// TwinCAT 3 PLC project PLC_LocateEdge
// ProgramVersion: 3.1.4023.0
// libraries:
//   Tc2_Standard, * (Beckhoff Automation GmbH)
//   Tc2_System, * (Beckhoff Automation GmbH)
//   Tc2_Utilities, * (Beckhoff Automation GmbH)
//   Tc3_Module, * (Beckhoff Automation GmbH)
//   Tc3_Vision, * (Beckhoff Automation GmbH)
// project tree:
//   DUTs/ ST_DimBase.TcDUT
//   GVLs/ GVL.TcGVL
//   / PlcTask.TcTTO, Vision_Job_Task_0.TcTTO
//   POUs/ FB_Camera.TcPOU, FB_MinAvgMax.TcPOU, F_Angle.TcPOU, F_Distance.TcPOU, F_DimDraw.TcPOU, MAIN.TcPOU, MAIN_VISION.TcPOU
// real-time tasks:
//   TASK PlcTask: cycle T#2ms, priority 4, ADS port 351
//   TASK VnTask ImgAcq (FileSource1): cycle T#5ms, priority 8, ADS port 350
//   TASK Vision Job Task 1: cycle default, priority 1
//   TASK Vision Job Task 0: cycle T#200000us, priority 10, ADS port 352

CONFIGURATION PLC_LocateEdge
    RESOURCE PLC ON TwinCAT3
        TASK PlcTask(INTERVAL := T#2ms, PRIORITY := 4);
        TASK Vision_Job_Task_0(INTERVAL := T#200000us, PRIORITY := 10);
        PROGRAM MAIN WITH PlcTask : MAIN;
        PROGRAM MAIN_VISION WITH Vision_Job_Task_0 : MAIN_VISION;
    END_RESOURCE
END_CONFIGURATION

// ---- DUTs/ST_DimBase.TcDUT
TYPE ST_DimBase :
STRUCT
	// Config
	name : STRING(255);
	
	// Must be set. Default values will return errors
	pFrom : TcVnPoint2_REAL := [-1, -1];
	pTo1 : TcVnPoint2_REAL := [-1, -1];
	pTo2 : TcVnPoint2_REAL := [-1, -1]; // Used for angle
	lines : UDINT := 0;
	
	// Can use defaults
	dir : ETcVnEdgeDirection := TCVN_ED_LIGHT_TO_DARK;
	minStr : REAL := 50;
	lineDist : REAL := 1;
	maxThick : UDINT := 10;
	gap : REAL := 0;
	precision : REAL := 0.0001; // 0.01 - 0.0001 only used for ERF/Gaussian
	subpix : UDINT := 1000; // 5-20 for INTER, 50-100 for ERF/Gaussian
	invDir : BOOL := FALSE;
	algorithm : ETcVnEdgeDetectionAlgorithm := TCVN_EDA_APPROX_ERF;
	degrees : BOOL := TRUE; // Used for angle
	
	// Results
	result : REAL;
	et : DINT; // Elapsed time in us
	complete : UDINT;
	results : ITcVnContainer; // Used for distance
	edgeFrom : ITcVnContainer;
	edgeTo : ITcVnContainer;
	lineFrom : TcVnVector4_LREAL;
	lineTo : TcVnVector4_LREAL;
END_STRUCT
END_TYPE

// ---- GVLs/GVL.TcGVL
VAR_GLOBAL
	camera : FB_Camera;
	dimDist : ARRAY [0..4] OF ST_DimBase := [
		(name:='d201', pFrom:=[115, 1290], pTo1:=[640, 1290], gap:=-1, lines:=291, lineDist:=3),
		(name:='d209', pFrom:=[245, 795], pTo1:=[245, 1770], gap:=-1, lines:=49, lineDist:=4),
		(name:='d222', pFrom:=[760, 875], pTo1:=[760, 1700], gap:=-1, lines:=45, lineDist:=4),
		(name:='od', pFrom:=[2260, 970], pTo1:=[2260, 1650], gap:=-1, lines:=121, lineDist:=4),
		(name:='gripper', pFrom:=[860, 450], pTo1:=[1850, 450], gap:=-1, lines:=161, lineDist:=5)
	];
END_VAR

// ---- POUs/MAIN.TcPOU
PROGRAM MAIN
VAR
	res : ARRAY [0..4] OF FB_MinAvgMax;
	ets : ARRAY [0..5] OF FB_MinAvgMax;
	total_et : DINT;
	test: BOOL;
	ii: INT;
	state: INT;
	cnt : INT;
	test2: BOOL;
	
	avg : LREAL;
	avg1 : TcVnVector2_LREAL;
	avg2 : TcVnVector2_LREAL;
	size1 : ULINT;
	size2 : ULINT;
	size3 : ULINT;
	
	idx : INT;
	arr1 : ARRAY [0..500] OF TcVnVector2_REAL;
	arr2 : ARRAY [0..500] OF TcVnVector2_REAL;
	arr3 : ARRAY [0..500] OF REAL;
END_VAR


IF test THEN
	test := FALSE;
	camera.trig();
END_IF

IF test2 THEN
	test2 := FALSE;
	F_VN_ContainerAverage(dimDist[idx].results, avg, S_OK);
	F_VN_ContainerAverageElementwise2(dimDist[idx].edgeFrom, avg1, S_OK);
	F_VN_ContainerAverageElementwise2(dimDist[idx].edgeTo, avg2, S_OK);
	
	F_VN_ExportContainerSize(dimDist[idx].edgeFrom, size1, S_OK);
	F_VN_ExportContainerSize(dimDist[idx].edgeTo, size2, S_OK);
	F_VN_ExportContainerSize(dimDist[idx].results, size3, S_OK);
	
	F_VN_ExportContainer(dimDist[idx].edgeFrom, ADR(arr1), SIZEOF(arr1), s_ok);
	F_VN_ExportContainer(dimDist[idx].edgeTo, ADR(arr2), SIZEOF(arr2), s_ok);
	F_VN_ExportContainer(dimDist[idx].results, ADR(arr3), SIZEOF(arr3), s_ok);
END_IF

CASE state OF
	10:
		camera.trig();
		state := 11;
	11:
		IF NOT camera.busy THEN
			total_et := 0;
			FOR ii := 0 TO 4 DO
				res[ii](IN:=dimDist[ii].result);
				ets[ii](IN:=dimDist[ii].et);
				total_et := total_et + dimDist[ii].et;
			END_FOR
			ets[5](IN:=total_et);
			cnt := cnt + 1;
			IF cnt < 100 THEN
				state := 10;
			ELSE
				cnt := 0;
				state := 0;
			END_IF
		END_IF
	12:
		FOR ii := 0 TO 4 DO
			res[ii].reset();
			ets[ii].reset();
		END_FOR
		ets[5].reset();
		state := 0;
END_CASE

END_PROGRAM

// ---- POUs/FB_MinAvgMax.TcPOU
FUNCTION_BLOCK FB_MinAvgMax
VAR_INPUT
	IN		: LREAL;
END_VAR
VAR_OUTPUT
	mini	: LREAL := 1.7976931348623158E308;
	avge	: LREAL;
	maxi	: LREAL := -1.7976931348623158E308;
END_VAR
VAR
	nums	: LREAL;
END_VAR

IF IN > maxi THEN
	maxi := IN;
END_IF
IF IN < mini THEN
	mini := IN;
END_IF

nums := nums + 1;
avge := avge + (IN - avge) / nums;

METHOD reset : BOOL
VAR_INPUT
END_VAR

mini := +1.7976931348623158E308;
maxi := -1.7976931348623158E308;
avge := 0;
nums := 0;
END_METHOD

END_FUNCTION_BLOCK

// ---- POUs/MAIN_VISION.TcPOU
PROGRAM MAIN_VISION
VAR
END_VAR


camera(dims := dimDist);

END_PROGRAM

// ---- POUs/FB_Camera.TcPOU
FUNCTION_BLOCK FB_Camera
VAR_IN_OUT
	dims : ARRAY [*] OF ST_DimBase;
END_VAR
VAR_OUTPUT
	busy : BOOL;
	ET : DINT;
END_VAR
VAR
	hr : HRESULT;
	hrFunc : HRESULT;
	hrWD : HRESULT;
	
	camera : FB_VN_SimpleCameraControl;
	camState : ETcVnCameraState;
	
	imgIn : ITcVnImage;
	imgInDisp : ITcVnDisplayableImage;
	imgOut : ITcVnImage;
	imgOutDisp : ITcVnDisplayableImage;
	
	state : INT;
	preempt : DINT;
	remain : DINT;
	complete : UDINT;
	ii : DINT;
	upper : DINT;
	lower : DINT;
	trigger : BOOL;
	cycleCnt : INT;
	old: INT;
	hr1:HRESULT;
	hr2:HRESULT;
END_VAR


camState := camera.GetState();
CASE state OF
	0:
		lower := LOWER_BOUND(dims, 1);
		upper := UPPER_BOUND(dims, 1);
		// Allow 1 ms for other items in task before and after vision
		preempt := TO_DINT(_TaskInfo[GETCURTASKINDEXEX()].CycleTime / 10) - 1000;
		IF preempt < 1000 THEN
			// Task cycle time is 1ms or less. Will not work.
			state := -1;
		ELSE
			state := 1000;
		END_IF
	1000:
		busy := FALSE;
		CASE camState OF
			TCVN_CS_INITIAL, TCVN_CS_OPENING, TCVN_CS_OPENED, TCVN_CS_STARTACQUISITION:
				hr := camera.StartAcquisition();
			TCVN_CS_Error:
				state := -1;
		END_CASE
	1010:
		CASE camState OF
			TCVN_CS_TRIGGERING:
				// If getting 16#98110712 the source likely has trigger disabled
				hr1 := camera.TriggerImage();
			TCVN_CS_ACQUIRING:
				IF trigger THEN
					hr2 := camera.TriggerImage();
					IF succeeded(hr2) THEN
						trigger := FALSE;
					END_IF
				ELSE
					hr := camera.GetCurrentImage(imgIn);
					IF SUCCEEDED(hr) AND_THEN imgIn <> 0 THEN
						ii := lower;
						ET := 0;
						cycleCnt := 0;
						state := 1020;
					END_IF
				END_IF
			TCVN_CS_ERROR:
				state := -1;
		END_CASE
	1020:
		remain := preempt; // Reset remain on each new cycle
		cycleCnt := cycleCnt + 1;
		FOR ii := ii TO upper DO
			hrWD := F_VN_StartRelWatchdog(remain, S_OK);
			// If returns 16#71A Task Watchdog Stack not enabled
			IF dims[ii].pTo2[0] = -1 THEN
				// pTo2 not used in Distance measurement
				hrFunc := F_Distance(dims[ii], imgIn);
			ELSE
				// But it is used in angle measurement
				hrFunc := F_Angle(dims[ii], imgIn);
			END_IF
			hrWD := F_VN_StopWatchdog(hrWD, nFractionProcessed=>complete, tRest=>remain);
			IF FAILED(hrFunc) OR_ELSE FAILED(hrWD) THEN
				// Send failed message
				// Will move on to other inspections and this one is ignored
			END_IF
			dims[ii].et := (cycleCnt * preempt) - ET - remain;
			dims[ii].complete := complete;
			ET := ET + dims[ii].et;
			IF complete <> 100 AND_THEN SUCCEEDED(hrFunc) THEN
				// Try calculation again in new cycle if not complete, but also not errored
				// Watchdog likely stopped it before completion
				EXIT;
			ELSIF ii = upper THEN
				// All calculations completed
				state := 1030;
				EXIT;
			ELSIF dims[ii+1].et > remain OR_ELSE (dims[ii+1].et = 0 AND_THEN remain < 1000) THEN
				// If the calculation was already done check its elapsed time larger than remain
				// If first time doing then try if more then 1ms remain otherwise start on new cycle
				ii := ii + 1;
				EXIT;
			END_IF
		END_FOR
	1030:
		hr := F_VN_ConvertColorSpace(imgIn, imgOut, TCVN_CST_GRAY_TO_RGB, hr);
		FOR ii := lower TO upper DO
			F_DimDraw(dims[ii], imgOut);
		END_FOR
		
		hr := F_VN_TransformIntoDisplayableImage(imgIn, imgInDisp, S_OK);
		hr := F_VN_TransformIntoDisplayableImage(imgOut, imgOutDisp, S_OK);
		state := 1000;
	-1000:
		// If stays in error then not linked to file/device
		// Check instance symbol initialization
		camera.Reset();
		IF camState <> TCVN_CS_ERROR THEN
			state := 0;
		END_IF
END_CASE

METHOD trig : BOOL
VAR_INPUT
END_VAR

IF state = 1000 AND_THEN camState = TCVN_CS_ACQUIRING AND_THEN NOT busy THEN
	busy := TRUE;
	ET := 0;
	trigger := TRUE;
	state := 1010;
END_IF
END_METHOD

END_FUNCTION_BLOCK

// ---- POUs/F_Distance.TcPOU
FUNCTION F_Distance : HRESULT
VAR_INPUT
	dim : REFERENCE TO ST_DimBase;
	img : ITcVnImage;
END_VAR


IF dim.gap < 0 THEN
	// If gap less than zero auto calculate based on largest diff between x/y and set to 80%
	// Helps reduce computation time
	dim.gap := MAX(ABS(dim.pTo1[0] - dim.pFrom[0]), ABS(dim.pTo1[1] - dim.pFrom[1])) * 0.8;
END_IF

F_Distance := F_VN_MeasureEdgeDistanceExp(
	ipSrcImage:=img,
	fAvgDistance:=dim.result,
	aStartPoint:=dim.pFrom,
	aEndPoint:=dim.pTo1,
	eEdgeDirection:=dim.dir,
	fMinStrength:=dim.minStr,
	nSearchLines:=dim.lines,
	fSearchLineDist:=dim.lineDist,
	nMaxThickness:=dim.maxThick,
	bInvertSearchDirection:=dim.invDir,
	fSearchGap:=dim.gap,
	nSubpixelsIterations:=dim.subpix,
	fApproxPrecision:=dim.precision,
	eAlgorithm:=dim.algorithm,
	ipEdgePoints1:=dim.edgeFrom,
	ipEdgePoints2:=dim.edgeTo,
	ipDistances:=dim.results,
	hrPrev:=S_OK
);

END_FUNCTION

// ---- POUs/F_Angle.TcPOU
FUNCTION F_Angle : HRESULT
VAR_INPUT
	dim : REFERENCE TO ST_DimBase;
	img : ITcVnImage;
END_VAR


F_Angle := F_VN_MeasureAngleBetweenEdgesExp(
	ipSrcImage:= img,
	fAngle:= dim.result,
	aInnerPoint:= dim.pFrom,
	aOuterPoint1:= dim.pTo1,
	aOuterPoint2:= dim.pTo2,
	eEdgeDirection:= dim.dir,
	fMinStrength:= dim.minStr,
	nSearchLines:= dim.lines,
	fSearchLineDist:= dim.lineDist,
	nMaxThickness:= dim.maxThick,
	bInvertSearchDirection:= dim.invDir,
	nSubpixelsIterations:= dim.subpix,
	bAngleInDegrees:= dim.degrees,
	fApproxPrecision:= dim.precision,
	eAlgorithm:= dim.algorithm,
	ipEdgePoints1:= dim.edgeFrom,
	ipEdgePoints2:= dim.edgeTo,
	hrPrev:=S_OK
);

END_FUNCTION

// ---- POUs/F_DimDraw.TcPOU
FUNCTION F_DimDraw : HRESULT
VAR_INPUT
	dim : REFERENCE TO ST_DimBase;
	img : ITcVnImage;
END_VAR
VAR
	hr : HRESULT;
	green : TcVnVector4_LREAL := [0, 255, 0, 0];
	blue : TcVnVector4_LREAL := [0, 0, 255, 0];
	red : TcVnVector4_LREAL := [255, 0, 0, 0];
END_VAR


IF dim.pFrom[0] >= 0 AND_THEN dim.pFrom[1] >= 0 THEN
	hr := F_VN_DrawPoint(TO_UDINT(dim.pFrom[0]), TO_UDINT(dim.pFrom[1]), img, TCVN_DS_CIRCLE, red, hr);
END_IF
IF dim.pTo1[0] >= 0 AND_THEN dim.pTo1[1] >= 0 THEN
	hr := F_VN_DrawPoint(TO_UDINT(dim.pTo1[0]), TO_UDINT(dim.pTo1[1]), img, TCVN_DS_X, red, hr);
END_IF
IF dim.pTo2[0] >= 0 AND_THEN dim.pTo2[1] >= 0 THEN
	hr := F_VN_DrawPoint(TO_UDINT(dim.pTo2[0]), TO_UDINT(dim.pTo2[1]), img, TCVN_DS_X, red, hr);
END_IF

IF F_VN_CheckIfEmpty(dim.edgeFrom, S_OK) = S_FALSE THEN
	hr := F_VN_DrawPointsExp(dim.edgeFrom, img, TCVN_DS_PLUS, blue, 1, 1, TCVN_LT_8_CONNECTED, hr);
	hr := F_VN_FitLine(dim.edgeFrom, dim.lineFrom, hr);
	hr := F_VN_DrawLine_TcVnVector4_LREAL(dim.lineFrom, img, green, 1, hr);
END_IF

IF F_VN_CheckIfEmpty(dim.edgeTo, S_OK) = S_FALSE THEN
	hr := F_VN_DrawPointsExp(dim.edgeTo, img, TCVN_DS_PLUS, blue, 1, 1, TCVN_LT_8_CONNECTED, hr);
	hr := F_VN_FitLine(dim.edgeTo, dim.lineTo, hr);
	hr := F_VN_DrawLine_TcVnVector4_LREAL(dim.lineTo, img, green, 1, hr);
END_IF
	
F_DimDraw := hr;

END_FUNCTION
